// TwinCAT 3 PLC project PLC1
// ProgramVersion: 3.1.4024.0
// libraries:
//   Tc2_Standard, * (Beckhoff Automation GmbH)
//   Tc2_System, * (Beckhoff Automation GmbH)
//   Tc3_Module, * (Beckhoff Automation GmbH)
// project tree:
//   / PlcTask.TcTTO
//   POUs/ MAIN.TcPOU
// real-time tasks:
//   TASK PlcTask: cycle T#10ms, priority 20, ADS port 350
// I/O:
//   DEVICE Device 1 (EtherCAT Automation Protocol), AmsNetId 192.168.10.20.2.1
//     Box 1 (Publisher)
//     Box 2 (Subscriber)
// variable links:
//   PLC1/PLC1 Instance <-> Device 1 (EtherCAT Automation Protocol)
//     PlcTask Inputs/MAIN.eap_state <-> Inputs/DevState
//   PLC1/PLC1 Instance <-> Device 1 (EtherCAT Automation Protocol)/Box 1 (Publisher)
//     PlcTask Outputs/MAIN.pub_bytes <-> RS1_Pub_Bytes/Outputs/VarData
//   PLC1/PLC1 Instance <-> Device 1 (EtherCAT Automation Protocol)/Box 2 (Subscriber)
//     PlcTask Inputs/MAIN.sub_bools <-> RS1_Sub_Bools/Inputs/VarData

CONFIGURATION PLC1
    RESOURCE PLC ON TwinCAT3
        TASK PlcTask(INTERVAL := T#10ms, PRIORITY := 20);
        PROGRAM MAIN WITH PlcTask : MAIN;
    END_RESOURCE
END_CONFIGURATION

// ---- POUs/MAIN.TcPOU
PROGRAM MAIN
VAR
	eap_state AT %I* : UINT;
	pub_bytes  AT %Q* :  ARRAY[0..19] OF BYTE;
	sub_bools  AT %I* :  ARRAY[0..9] OF BOOL;
END_VAR

END_PROGRAM
